// TIA Portal V17 export
// export: Created 2023-02-13T11:16:55.9412334Z, ExportSetting WithDefaults, DisplayName Totally Integrated Automation Portal, DisplayVersion V17, DisplayName TIA Portal Openness, DisplayVersion V17, DisplayName TIA Portal Teamcenter Gateway, DisplayVersion V17, DisplayName TIA Portal Version Control Interface, DisplayVersion V17, DisplayName SINAMICS Startdrive Advanced, DisplayVersion V17, DisplayName SINAMICS Startdrive G130, G150, S120, S150, SINAMICS MV, S210, DisplayVersion V17, DisplayName SINAMICS Startdrive G110M, G120, G120C, G120D, G120P, G115D, DisplayVersion V17, DisplayName STEP 7 Professional, DisplayVersion V17, DisplayName STEP 7 Safety, DisplayVersion V17, DisplayName WinCC Professional, DisplayVersion V17
DATA_BLOCK "T-31.00_DB"   // DB25
VERSION : 0.1
// stored: AutoNumber true, DBAccessibleFromOPCUA true, DBAccessibleFromWebserver true, InstanceOfName BLEND, InstanceOfType FB
"BLEND"
   // VAR_INPUT
   //    Lock : Bool;
   //    Reset : Bool;
   //    ENTransfer : Bool;
   //    ENProd : Bool;
   //    THE_ProdReq : Bool;
   //    THE_ProdLineOpen : Bool;
   //    THE_CIPLineOpen : Bool;
   //    THE_CIP_En : Bool;
   //    MixproofFlip : Bool;
   //    FB_AV_Transfer : Bool;
   //    FB_P_Transfer : Bool;
   //    Level : Real;
   //    Temp : Real;
   //    TransfPump_AVSpeed : Real;
   // END_VAR
   // VAR_OUTPUT
   //    Q_Prod : Bool;
   //    Q_Trans : Bool;
   //    Q_CIPReq : Bool;
   //    Q_MixProofFlif : Bool;
   //    QAV_Transfer : Bool;
   //    QP_Transfer : Bool;
   // END_VAR
   // VAR
   //    Cmd : Struct
   //       Transfer_ON : Bool;
   //       Transfer_OFF : Bool;
   //    END_STRUCT;
   //    HMI : Struct
   //       Cmd : DWord;
   //       Cmd_EN : DWord;
   //       Cmd_Stat : DWord;
   //       MatSel : DWord;
   //       DoseStart : DWord;
   //       DosePause : DWord;
   //       DoseStop : DWord;
   //       DoseState : DWord;
   //    END_STRUCT;
   //    Tank_Par : Struct
   //       LL : Real;
   //       LB_OFF : Real;
   //       LB_ON : Real;
   //       LB1_OFF : Real;
   //       LB1_ON : Real;
   //       LB2_OFF : Real;
   //       LB2_ON : Real;
   //       LB3_OFF : Real;
   //       LB3_ON : Real;
   //       P01_ProdSP : Real;
   //       P01_CIPSP : Real;
   //    END_STRUCT;
   //    Tank_Sta : Struct
   //       LL : Bool;
   //       LB_OFF : Bool;
   //       LB_ON : Bool;
   //       LB1_OFF : Bool;
   //       LB1_ON : Bool;
   //       LB2_OFF : Bool;
   //       LB2_ON : Bool;
   //       LB3_OFF : Bool;
   //       LB3_ON : Bool;
   //       Agi_ON : Bool;
   //       TranferON : Bool;
   //       Inload : Bool;
   //       CIPRequest : Bool;
   //       AwysON : Bool;
   //    END_STRUCT;
   //    SP_Water : "RawDose";
   //    SP_Sugar { S7_SetPoint := 'True'} : "RawDose";
   //    SP_Garam { S7_SetPoint := 'True'} : "RawDose";
   //    SP_ChiliAwet_1 { S7_SetPoint := 'True'} : "RawDose";
   //    SP_ChiliAwet_2 { S7_SetPoint := 'True'} : "RawDose";
   //    SP_ChiliAwet_3 { S7_SetPoint := 'True'} : "RawDose";
   //    SP_ChiliFresh_1 { S7_SetPoint := 'True'} : "RawDose";
   //    SP_ChiliFresh_2 { S7_SetPoint := 'True'} : "RawDose";
   //    SP_ChiliFresh_3 { S7_SetPoint := 'True'} : "RawDose";
   //    SP_Garlic { S7_SetPoint := 'True'} : "RawDose";
   //    SP_Vinegar { S7_SetPoint := 'True'} : "RawDose";
   //    SP_Tomato { S7_SetPoint := 'True'} : "RawDose";
   //    SP_Homomix { S7_SetPoint := 'True'} : "RawDose";
   //    SP_Rework { S7_SetPoint := 'True'} : "RawDose";
   //    Water : "DOSE";
   //    Sugar { S7_SetPoint := 'True'} : "DOSE";
   //    Garam : "DOSE";
   //    ChiliAwet_1 { S7_SetPoint := 'True'} : "DOSE";
   //    ChiliAwet_2 { S7_SetPoint := 'True'} : "DOSE";
   //    ChiliAwet_3 { S7_SetPoint := 'True'} : "DOSE";
   //    ChiliFresh_1 { S7_SetPoint := 'True'} : "DOSE";
   //    ChiliFresh_2 { S7_SetPoint := 'True'} : "DOSE";
   //    ChiliFresh_3 { S7_SetPoint := 'True'} : "DOSE";
   //    Garlic { S7_SetPoint := 'True'} : "DOSE";
   //    Vinegar { S7_SetPoint := 'True'} : "DOSE";
   //    Tomato { S7_SetPoint := 'True'} : "DOSE";
   //    Homomix { S7_SetPoint := 'True'} : "DOSE";
   //    Rework { S7_SetPoint := 'True'} : "DOSE";
   //    RdyforTransfer : Struct
   //       cmd_on : Bool;
   //       cmd_off : Bool;
   //       EnCmd : Bool;
   //       Stat_ON : Bool;
   //       Stat_Stop : Bool;
   //    END_STRUCT;
   //    Transfer : Struct
   //       cmd_on : Bool;
   //       cmd_off : Bool;
   //       EnCmd : Bool;
   //       Stat_ON : Bool;
   //       Stat_Stop : Bool;
   //    END_STRUCT;
   //    CIP : Struct
   //       cmd_on : Bool;
   //       cmd_off : Bool;
   //       EnCmd : Bool;
   //       Stat_ON : Bool;
   //       Stat_Stop : Bool;
   //    END_STRUCT;
   //    Agitator : Struct
   //       cmd_on : Bool;
   //       cmd_off : Bool;
   //       EnCmd : Bool;
   //       Stat_ON : Bool;
   //       Stat_Stop : Bool;
   //    END_STRUCT;
   //    PumpOFFTimer : TON_TIME;
   //    TransitionTimer { S7_SetPoint := 'True'} : TON_TIME;
   // END_VAR
BEGIN
END_DATA_BLOCK
